Fanuc KAREL source: IO0067.KL

-- PROVISIONAL review KL for V770-1; original PC SHA256 3207a29265b58a6fa21a60459021ac939affac1f21dfa0d1b1255986325c0bbd
-- Incomplete behavior may be omitted. Consult companion uncertainty JSON. Do not deploy.
PROGRAM IO0067
%NOLOCKGROUP
-- UNRESOLVED_LOCAL_POOL 5 cells at code offset 13; source declarations unknown
-- DIRECT_LOCAL_WORD_ACCESS alone does not prove INTEGER, REAL, or BOOLEAN
BEGIN
  -- UNRESOLVED_PC offsets 0-18; opcodes 2B,2C,7B
  -- UNRESOLVED_PC offsets 23-30; opcodes 9D,23
  -- UNRESOLVED_PC offsets 35-49; opcodes 2E,22,9D,33,35
  -- UNRESOLVED_PC offsets 54-61; opcodes 9D,23
  -- UNRESOLVED_PC offsets 66-77; opcodes 2E,23
  -- UNRESOLVED_PC offsets 82-92; opcodes 9D,19,9C,5B,79
  -- UNRESOLVED_PC offsets 97-111; opcodes 21,9D,52,23
  -- UNRESOLVED_PC offsets 121-125; opcodes 7F
  -- UNRESOLVED_PC offsets 130-134; opcodes 27,AA
  -- UNRESOLVED_PC offsets 139-143; opcodes 7F
END IO0067
